TEXTLIST CtrlMode_List
  1 = 'Local Mode'
  2 = 'Remote Mode'
   = ''
END_TEXTLIST

(* stored: Version 1.1.0.1, ProductVersion 3.1.4018.5
   TextList CtrlMode_List: Id {d6ba1d83-6225-41c3-b5e1-76c46f971e29} *)
